FUNCTION_BLOCK FB_HotConnect2
VAR_INPUT
END_VAR
VAR_OUTPUT
END_VAR
VAR
END_VAR

END_FUNCTION_BLOCK

(* stored: Version 1.1.0.1, ProductVersion 3.1.4024.6
   POU FB_HotConnect2: Id {edf59865-9bbd-4e75-9a19-f5cf1e484e54}, SpecialFunc None *)
